Omron CX-Programmer project NewProject (CX-Programmer ?)

# PLC NewPLC1: CS1H CPU63

## Program MASTER (cyclic task 0)

### Section Section1

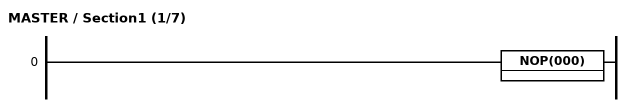
; rung 0
NOP(000)

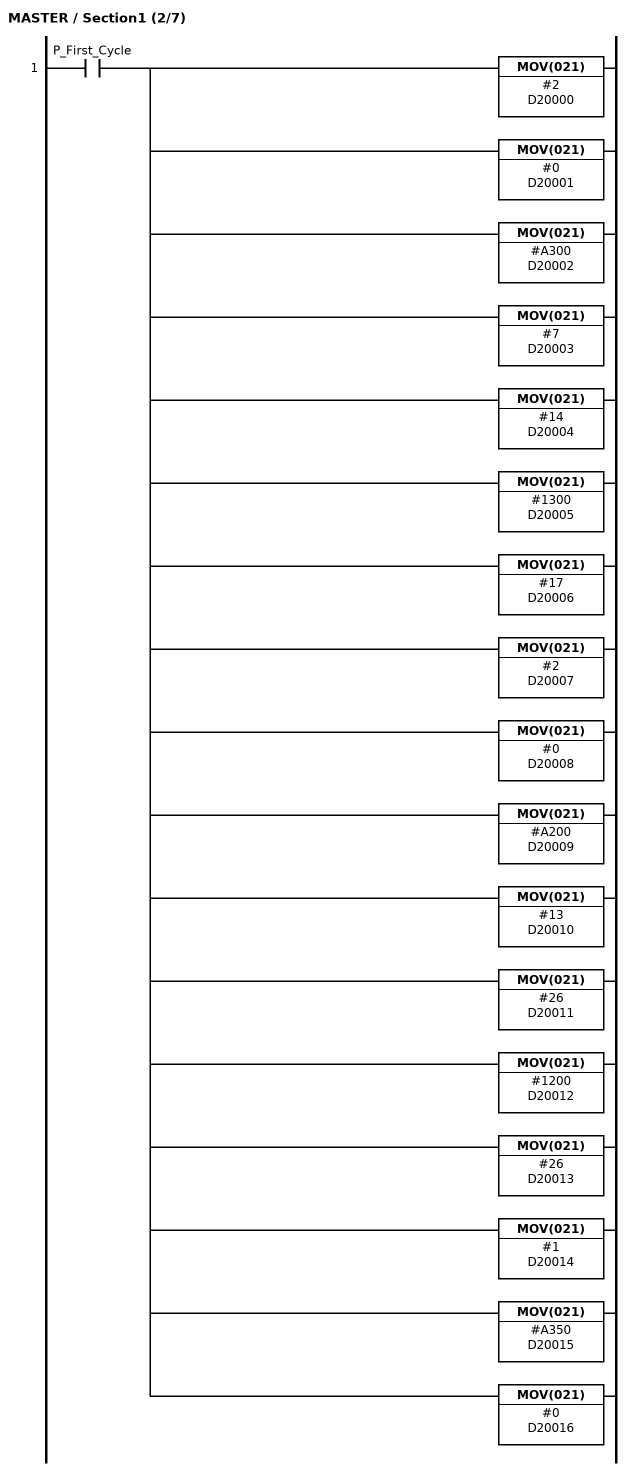
; rung 1
// R
LD P_First_Cycle  // 
MOV(021) #2 D20000
MOV(021) #0 D20001
MOV(021) #A300 D20002
MOV(021) #7 D20003
MOV(021) #14 D20004
MOV(021) #1300 D20005
MOV(021) #17 D20006
MOV(021) #2 D20007
MOV(021) #0 D20008
MOV(021) #A200 D20009
MOV(021) #13 D20010
MOV(021) #26 D20011
MOV(021) #1200 D20012
MOV(021) #26 D20013
MOV(021) #1 D20014
MOV(021) #A350 D20015
MOV(021) #0 D20016

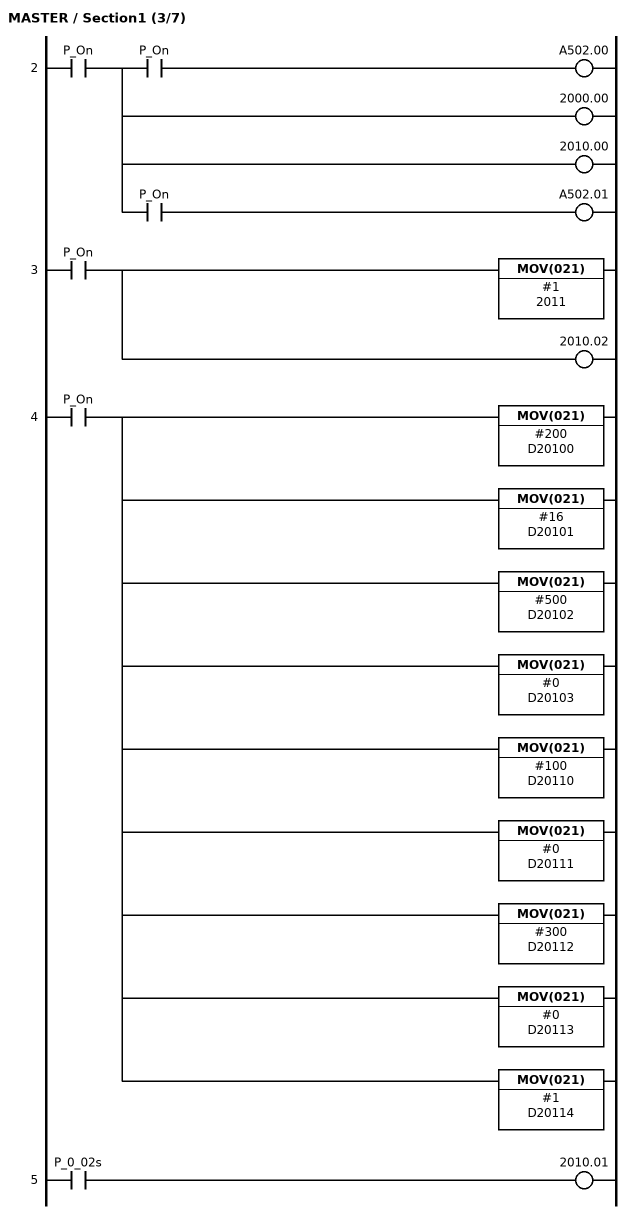
; rung 2
LD P_On
OUT TR0
AND P_On
OUT A502.00
LD TR0
OUT 2000.00
OUT 2010.00
AND P_On
OUT A502.01
; rung 3
LD P_On
MOV(021) #1 2011
OUT 2010.02
; rung 4
LD P_On
MOV(021) #200 D20100
MOV(021) #16 D20101
MOV(021) #500 D20102
MOV(021) #0 D20103
MOV(021) #100 D20110
MOV(021) #0 D20111
MOV(021) #300 D20112
MOV(021) #0 D20113
MOV(021) #1 D20114
; rung 5
LD P_0_02s
OUT 2010.01

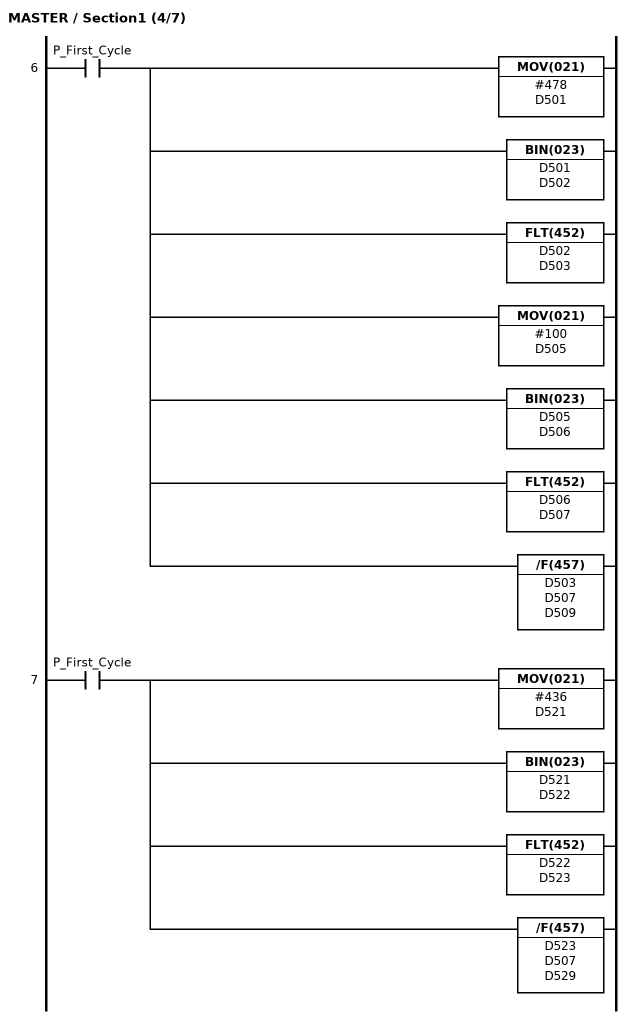
; rung 6
// R
LD P_First_Cycle
MOV(021) #478 D501
BIN(023) D501 D502
FLT(452) D502 D503
MOV(021) #100 D505
BIN(023) D505 D506
FLT(452) D506 D507
/F(457) D503 D507 D509  // 
; rung 7
// R
LD P_First_Cycle
MOV(021) #436 D521
BIN(023) D521 D522
FLT(452) D522 D523
/F(457) D523 D507 D529  // 

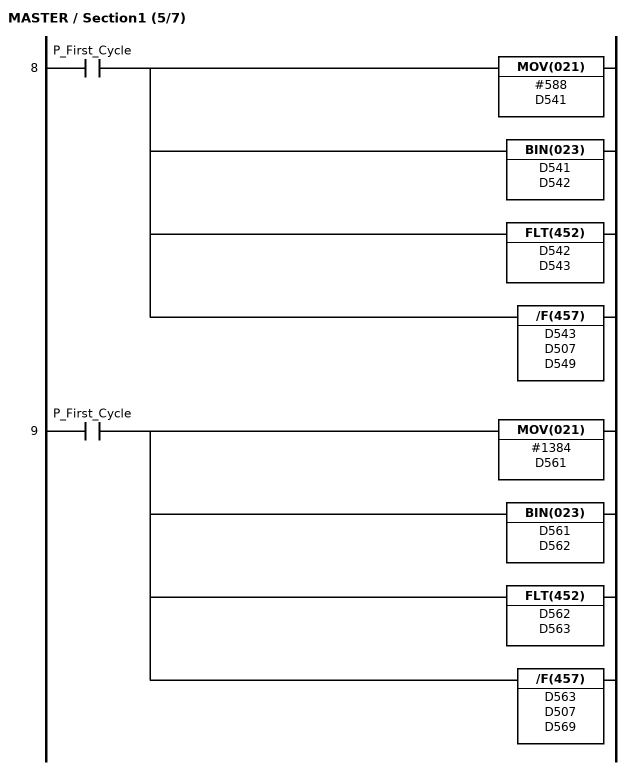
; rung 8
// R
LD P_First_Cycle
MOV(021) #588 D541
BIN(023) D541 D542
FLT(452) D542 D543
/F(457) D543 D507 D549  // 
; rung 9
// R
LD P_First_Cycle
MOV(021) #1384 D561
BIN(023) D561 D562
FLT(452) D562 D563
/F(457) D563 D507 D569  // 

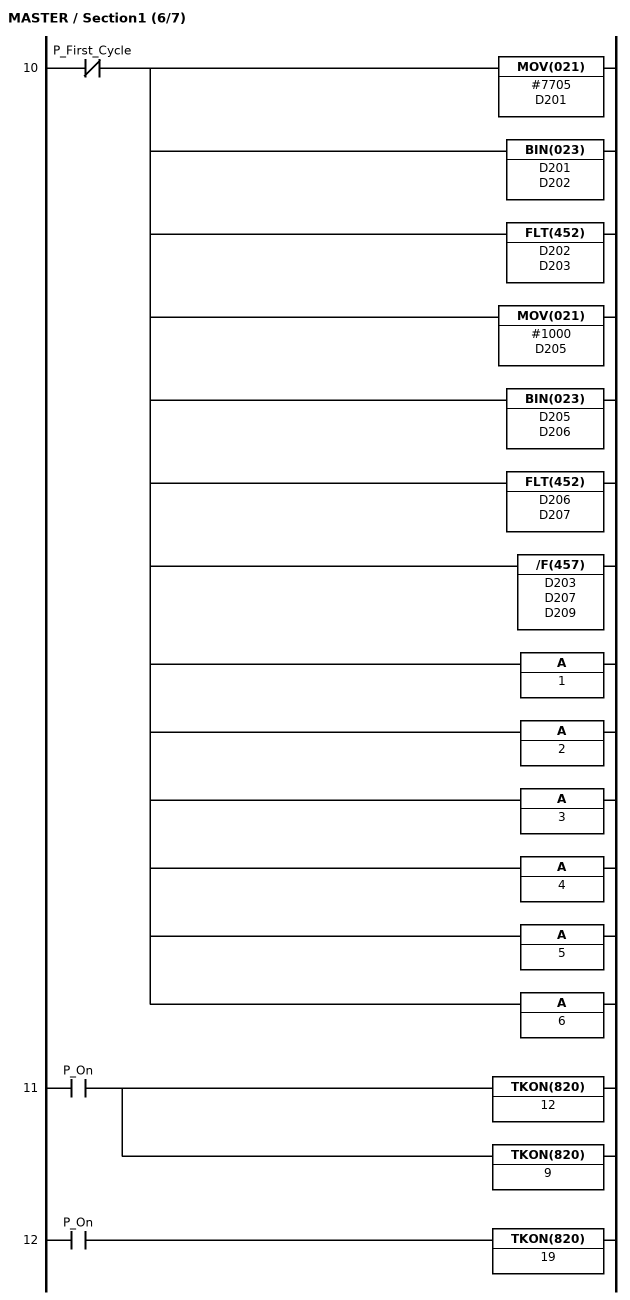
; rung 10
// R
LDNOT P_First_Cycle
MOV(021) #7705 D201
BIN(023) D201 D202
FLT(452) D202 D203
MOV(021) #1000 D205
BIN(023) D205 D206
FLT(452) D206 D207
/F(457) D203 D207 D209  // 
A  1
A  2
A  3
A  4
A  5
A  6
// 
// 
// 
// 
// 
// 
; rung 11
// R
LD P_On
TKON(820) 12
TKON(820) 9  // 
; rung 12
// R
LD P_On
TKON(820) 19  // 

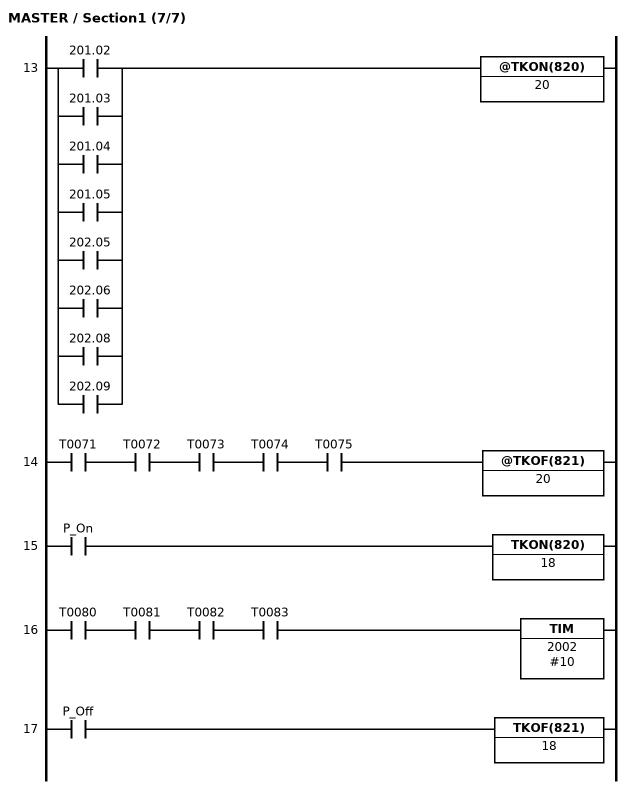
; rung 13
// R
LD 201.02
OR 201.03
OR 201.04
OR 201.05
OR 202.05
OR 202.06
OR 202.08
OR 202.09
@TKON(820) 20  // 
; rung 14
LD T0071
AND T0072
AND T0073
AND T0074
AND T0075
@TKOF(821) 20
; rung 15
// R
LD P_On
TKON(820) 18  // 
; rung 16
LD T0080
AND T0081
AND T0082
AND T0083
TIM 2002 #10
; rung 17
LD P_Off
TKOF(821) 18

### Section Section2

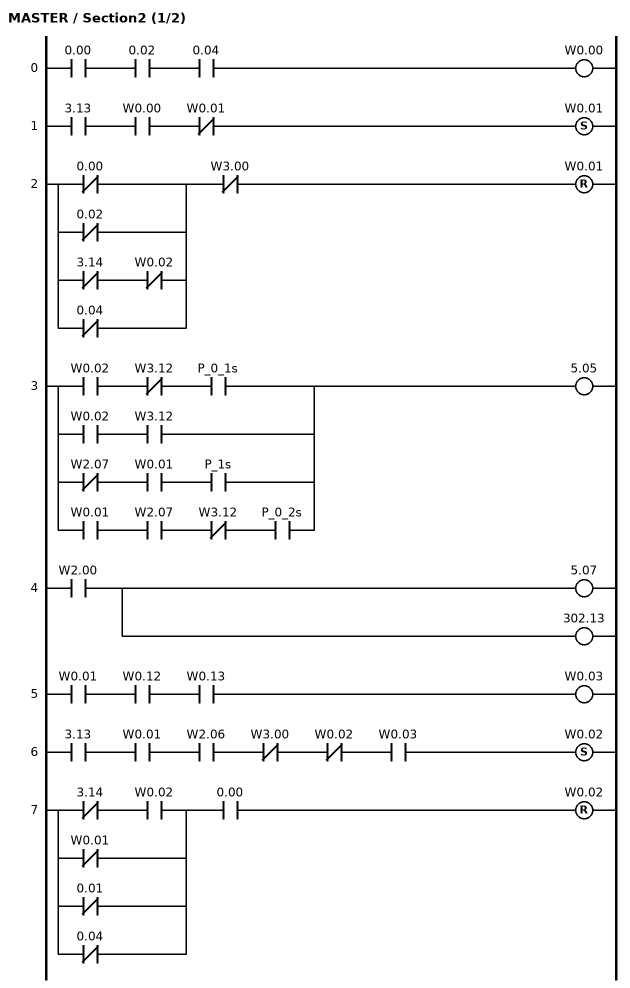
; rung 0
// R
LD 0.00
AND 0.02
AND 0.04
OUT W0.00  // 
; rung 1
LD 3.13
AND W0.00
ANDNOT W0.01
SET W0.01  // 
; rung 2
LDNOT 0.00
ORNOT 0.02
LDNOT 3.14
ANDNOT W0.02
ORLD
ORNOT 0.04
ANDNOT W3.00
RSET W0.01
; rung 3
LD W0.02
ANDNOT W3.12
AND P_0_1s
LD W0.02
AND W3.12
ORLD
LDNOT W2.07
AND W0.01
AND P_1s
ORLD
LD W0.01
AND W2.07
ANDNOT W3.12
AND P_0_2s
ORLD
OUT 5.05
; rung 4
LD W2.00
OUT 5.07
OUT 302.13
; rung 5
LD W0.01
AND W0.12
AND W0.13
OUT W0.03  // 
; rung 6
// R
LD 3.13
AND W0.01
AND W2.06
ANDNOT W3.00
ANDNOT W0.02
AND W0.03
SET W0.02
; rung 7
LDNOT 3.14
AND W0.02
ORNOT W0.01
ORNOT 0.01
ORNOT 0.04
AND 0.00
RSET W0.02

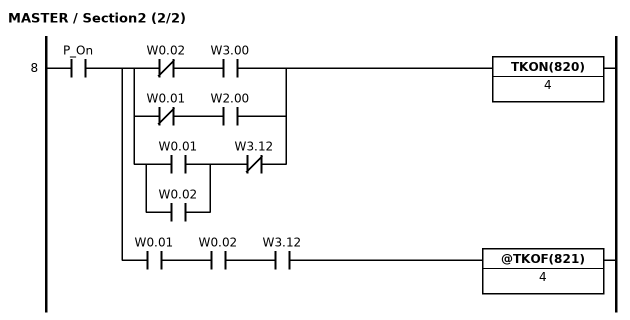
; rung 8
LD P_On
OUT TR0
LDNOT W0.02
AND W3.00
LDNOT W0.01
AND W2.00
ORLD
LD W0.01
OR W0.02
ANDNOT W3.12
ORLD
ANDLD
TKON(820) 4
LD TR0
AND W0.01
AND W0.02
AND W3.12
@TKOF(821) 4  // 

### Section Section3

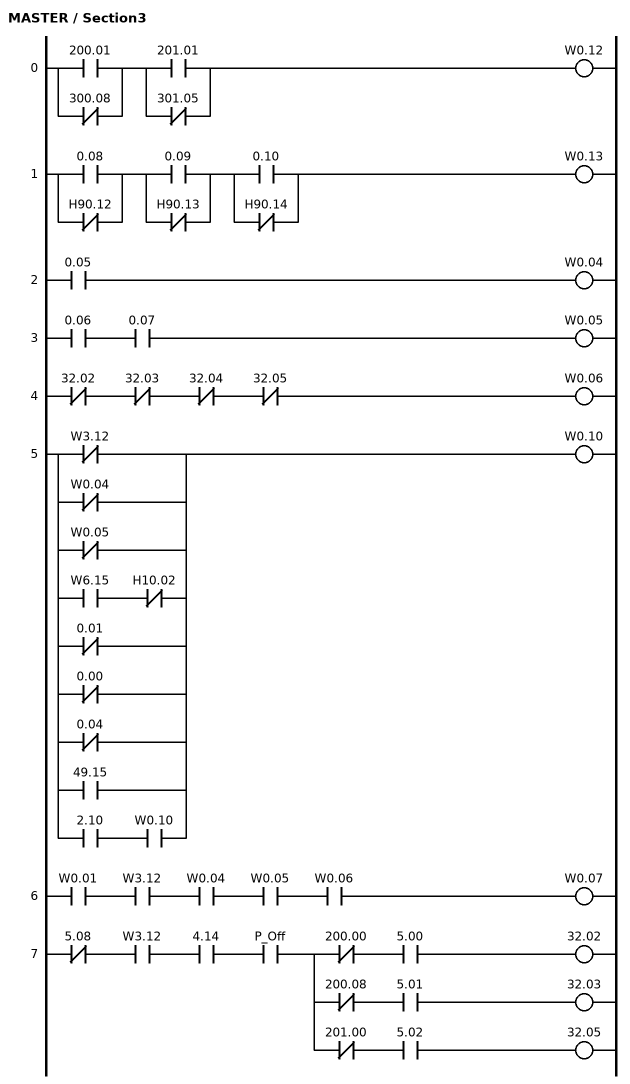
; rung 0
// R
LD 200.01
ORNOT 300.08
LD 201.01
ORNOT 301.05
ANDLD
OUT W0.12
; rung 1
LD 0.08
ORNOT H90.12
LD 0.09
ORNOT H90.13
ANDLD
LD 0.10
ORNOT H90.14
ANDLD
OUT W0.13
; rung 2
LD 0.05
OUT W0.04
; rung 3
LD 0.06
AND 0.07
OUT W0.05
; rung 4
LDNOT 32.02
ANDNOT 32.03
ANDNOT 32.04
ANDNOT 32.05
OUT W0.06
; rung 5
LDNOT W3.12
ORNOT W0.04
ORNOT W0.05
LD W6.15
ANDNOT H10.02
ORLD
ORNOT 0.01
ORNOT 0.00
ORNOT 0.04
OR 49.15
LD 2.10
AND W0.10
ORLD
OUT W0.10
; rung 6
LD W0.01
AND W3.12
AND W0.04
AND W0.05
AND W0.06
OUT W0.07
; rung 7
// R
LDNOT 5.08
AND W3.12
AND 4.14
AND P_Off
OUT TR0
ANDNOT 200.00
AND 5.00
OUT 32.02
LD TR0
ANDNOT 200.08
AND 5.01
OUT 32.03
LD TR0
ANDNOT 201.00
AND 5.02
OUT 32.05

### Section Section4

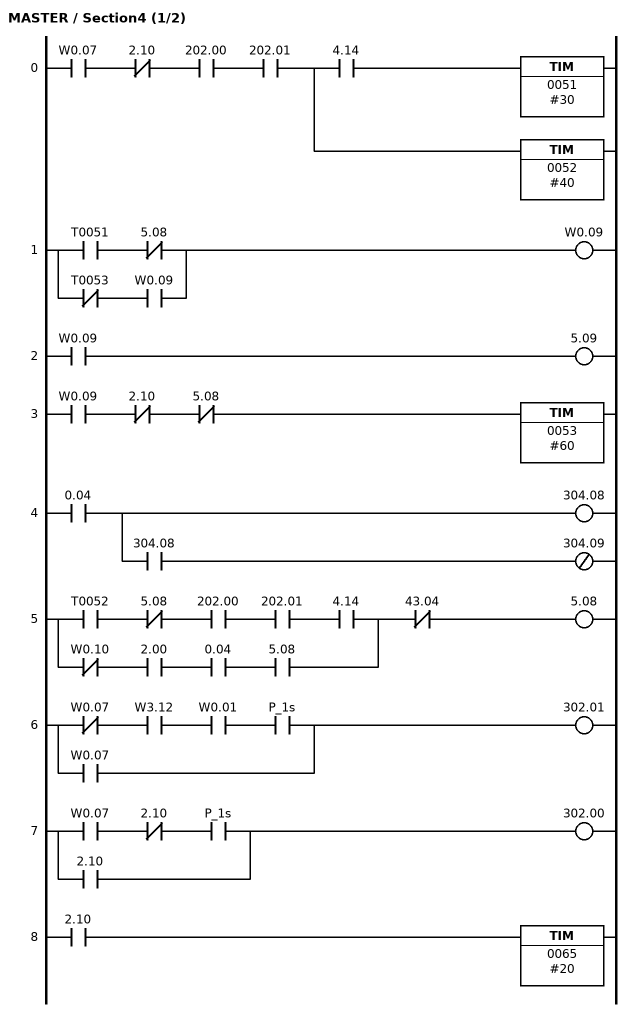
; rung 0
// R
LD W0.07
ANDNOT 2.10
AND 202.00
AND 202.01
OUT TR0
AND 4.14
TIM 0051 #30
LD TR0
TIM 0052 #40
; rung 1
LD T0051
ANDNOT 5.08
LDNOT T0053
AND W0.09
ORLD
OUT W0.09
; rung 2
LD W0.09
OUT 5.09
; rung 3
LD W0.09
ANDNOT 2.10
ANDNOT 5.08
TIM 0053 #60
; rung 4
LD 0.04
OUT 304.08
AND 304.08
OUTNOT 304.09
; rung 5
LD T0052
ANDNOT 5.08
AND 202.00
AND 202.01
AND 4.14
LDNOT W0.10
AND 2.00
AND 0.04
AND 5.08
ORLD
ANDNOT 43.04
OUT 5.08
; rung 6
LDNOT W0.07
AND W3.12
AND W0.01
AND P_1s
OR W0.07
OUT 302.01
; rung 7
LD W0.07
ANDNOT 2.10
AND P_1s
OR 2.10
OUT 302.00
; rung 8
LD 2.10
TIM 0065 #20

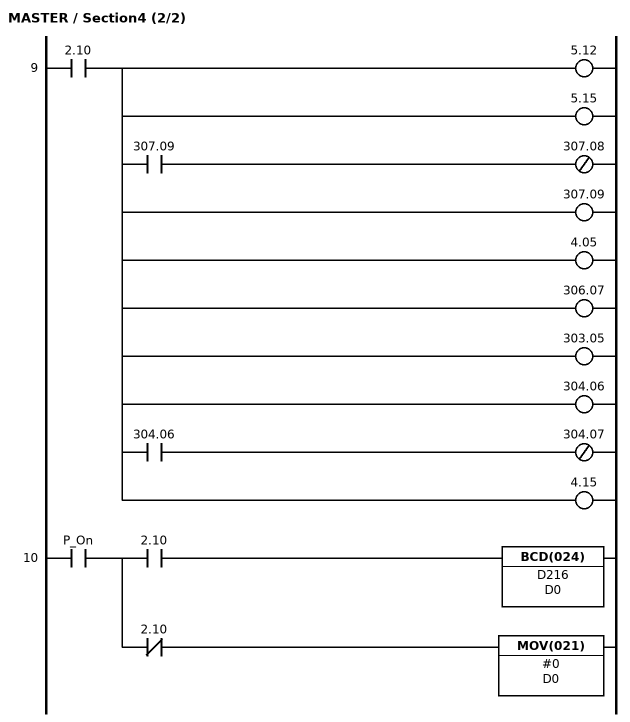
; rung 9
LD 2.10
OUT TR0
OUT 5.12
OUT 5.15
AND 307.09
OUTNOT 307.08
LD TR0
OUT 307.09
OUT 4.05
OUT 306.07
OUT 303.05
OUT 304.06
AND 304.06
OUTNOT 304.07
LD TR0
OUT 4.15
; rung 10
LD P_On
OUT TR0
AND 2.10
BCD(024) D216 D0
LD TR0
ANDNOT 2.10
MOV(021) #0 D0

### Section Section5

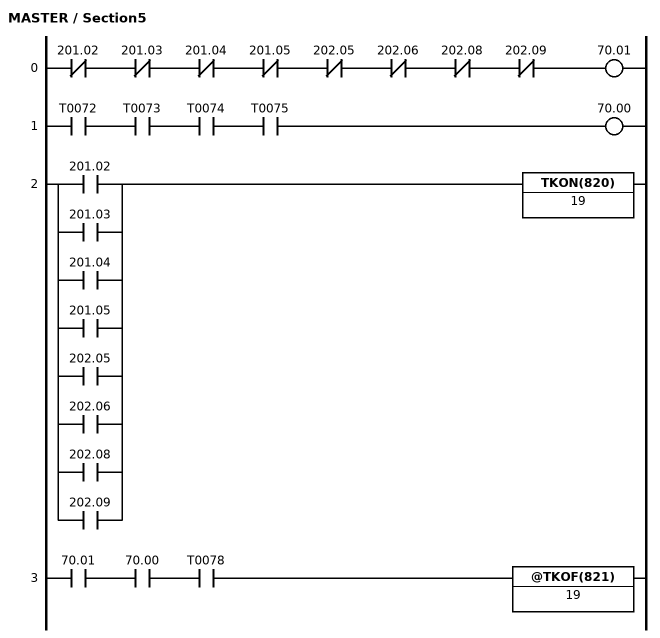
; rung 0
LDNOT 201.02
ANDNOT 201.03
ANDNOT 201.04
ANDNOT 201.05
ANDNOT 202.05
ANDNOT 202.06
ANDNOT 202.08
ANDNOT 202.09
OUT 70.01
; rung 1
LD T0072
AND T0073
AND T0074
AND T0075
OUT 70.00
; rung 2
LD 201.02
OR 201.03
OR 201.04
OR 201.05
OR 202.05
OR 202.06
OR 202.08
OR 202.09
TKON(820) 19  // 
; rung 3
LD 70.01
AND 70.00
AND T0078
@TKOF(821) 19

### Section Section6

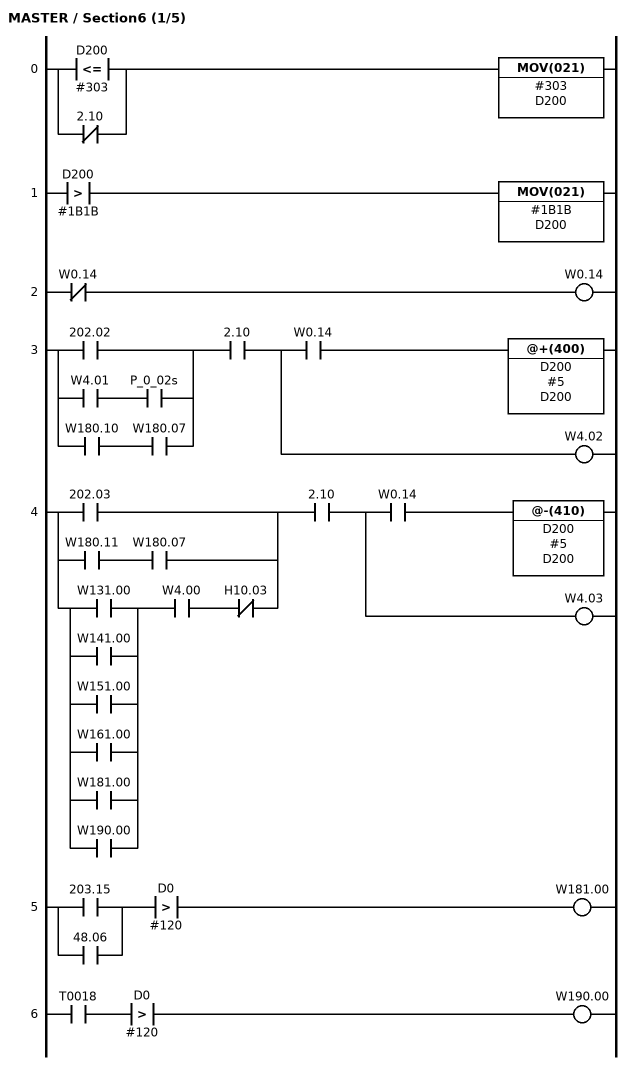
; rung 0
// R
LD<=(315) D200 #303
ORNOT 2.10
MOV(021) #303 D200  // 
; rung 1
LD>(320) D200 #1B1B
MOV(021) #1B1B D200  // 
; rung 2
LDNOT W0.14
OUT W0.14
; rung 3
// R
LD 202.02
LD W4.01
AND P_0_02s
ORLD
LD W180.10
AND W180.07
ORLD
AND 2.10
OUT TR0
AND W0.14
@+(400) D200 #5 D200
LD TR0
OUT W4.02  // 
; rung 4
// R
LD 202.03
LD W180.11
AND W180.07
ORLD
LD W131.00
OR W141.00
OR W151.00
OR W161.00
OR W181.00
OR W190.00
AND W4.00
ANDNOT H10.03
ORLD
AND 2.10
OUT TR0
AND W0.14
@-(410) D200 #5 D200
LD TR0
OUT W4.03  // 
; rung 5
// R
LD 203.15
OR 48.06
AND>(320) D0 #120
OUT W181.00
; rung 6
// R
LD T0018
AND>(320) D0 #120
OUT W190.00

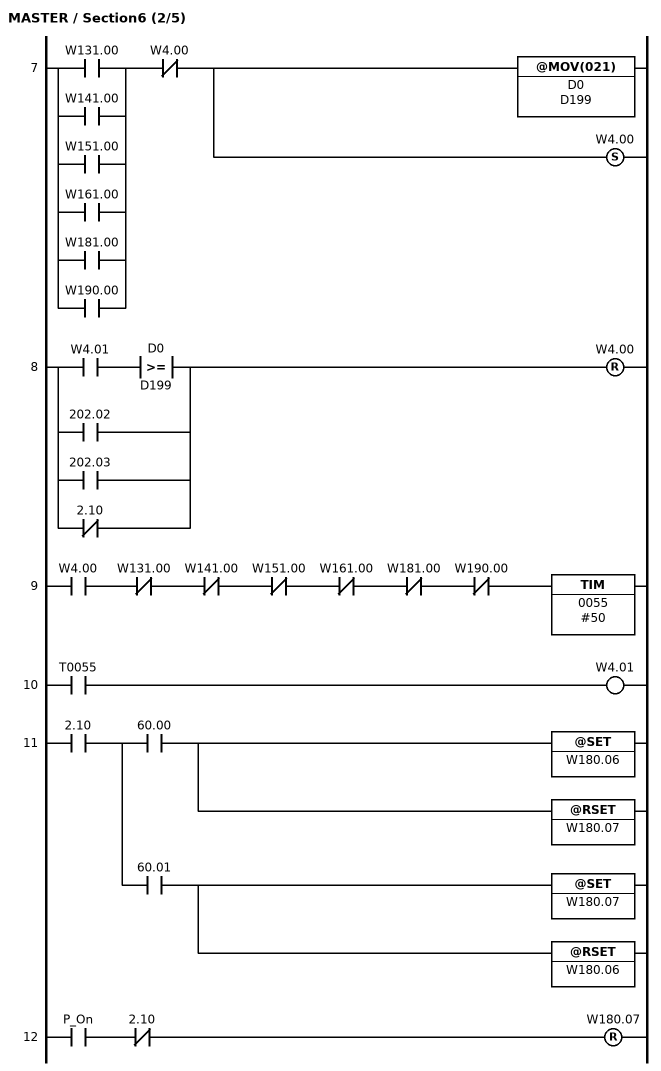
; rung 7
// R
LD W131.00
OR W141.00
OR W151.00
OR W161.00
OR W181.00
OR W190.00
ANDNOT W4.00
@MOV(021) D0 D199
SET W4.00
; rung 8
LD W4.01
AND>=(325) D0 D199
OR 202.02
OR 202.03
ORNOT 2.10
RSET W4.00
; rung 9
LD W4.00
ANDNOT W131.00
ANDNOT W141.00
ANDNOT W151.00
ANDNOT W161.00
ANDNOT W181.00
ANDNOT W190.00
TIM 0055 #50
; rung 10
LD T0055
OUT W4.01
; rung 11
LD 2.10
OUT TR0
AND 60.00
@SET W180.06
@RSET W180.07
LD TR0
AND 60.01
@SET W180.07
@RSET W180.06
; rung 12
LD P_On
ANDNOT 2.10
RSET W180.07

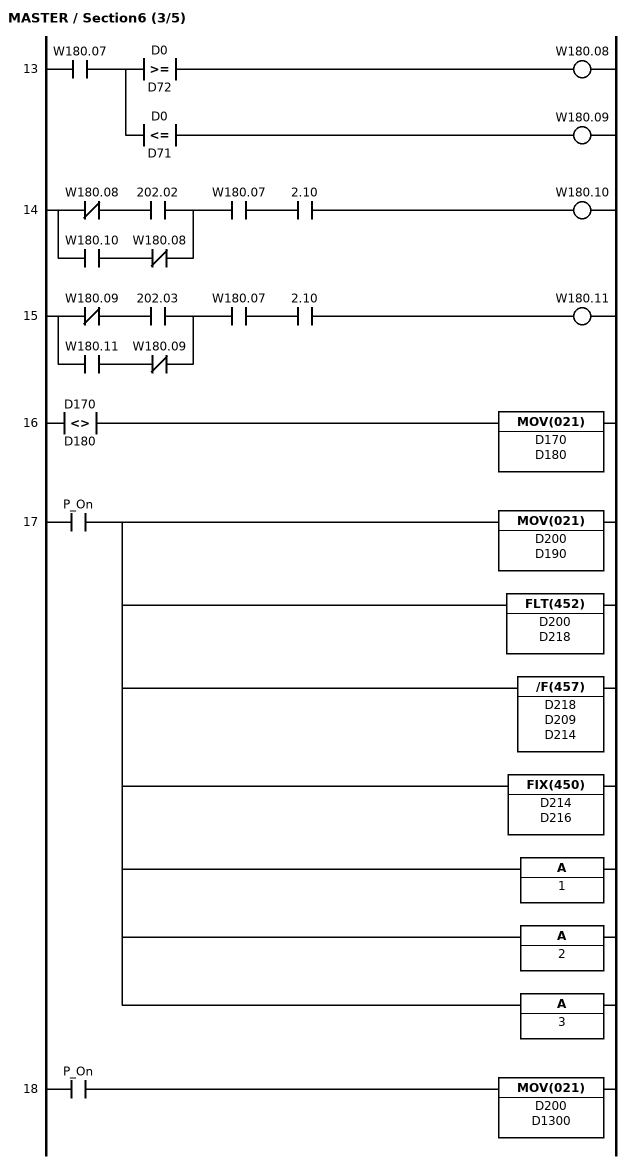
; rung 13
LD W180.07
OUT TR0
AND>=(325) D0 D72
OUT W180.08
LD TR0
AND<=(315) D0 D71
OUT W180.09
; rung 14
LDNOT W180.08
AND 202.02
LD W180.10
ANDNOT W180.08
ORLD
AND W180.07
AND 2.10
OUT W180.10
; rung 15
LDNOT W180.09
AND 202.03
LD W180.11
ANDNOT W180.09
ORLD
AND W180.07
AND 2.10
OUT W180.11
; rung 16
LD<>(305) D170 D180
MOV(021) D170 D180
; rung 17
// R
LD P_On
MOV(021) D200 D190
FLT(452) D200 D218
/F(457) D218 D209 D214
FIX(450) D214 D216  // 
A  1
A  2
A  3
// 
// 
// 
; rung 18
// R
LD P_On
MOV(021) D200 D1300

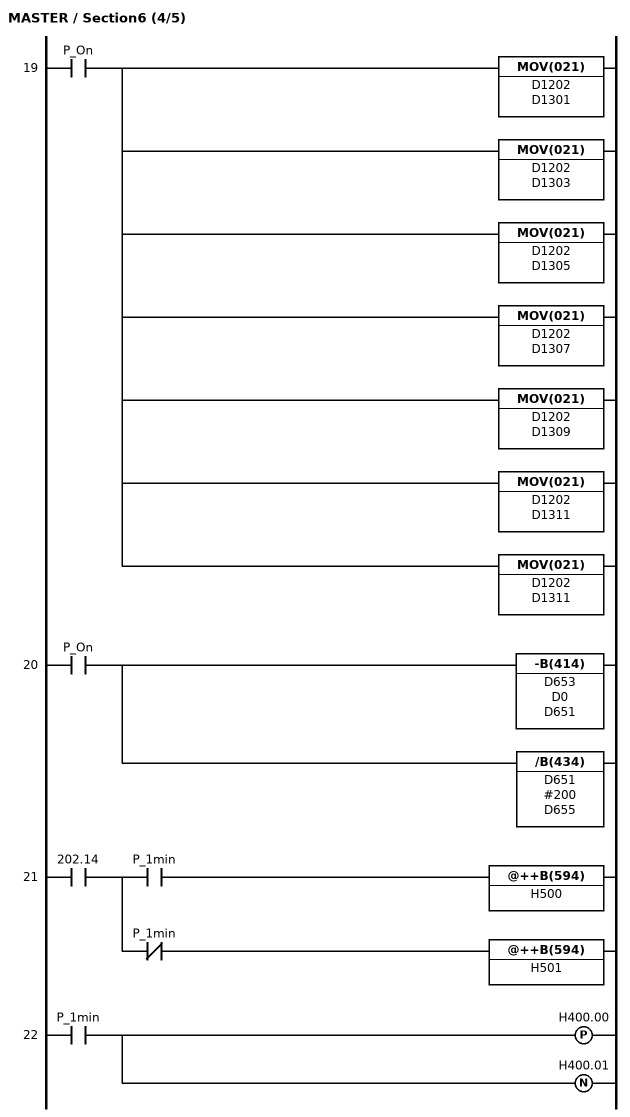
; rung 19
// R
LD P_On
MOV(021) D1202 D1301
MOV(021) D1202 D1303
MOV(021) D1202 D1305
MOV(021) D1202 D1307
MOV(021) D1202 D1309
MOV(021) D1202 D1311
MOV(021) D1202 D1311
; rung 20
LD P_On
-B(414) D653 D0 D651
/B(434) D651 #200 D655
; rung 21
// R
LD 202.14
OUT TR0
AND P_1min
@++B(594) H500
LD TR0
ANDNOT P_1min
@++B(594) H501
; rung 22
LD P_1min
DIFU(013) H400.00
DIFD(014) H400.01

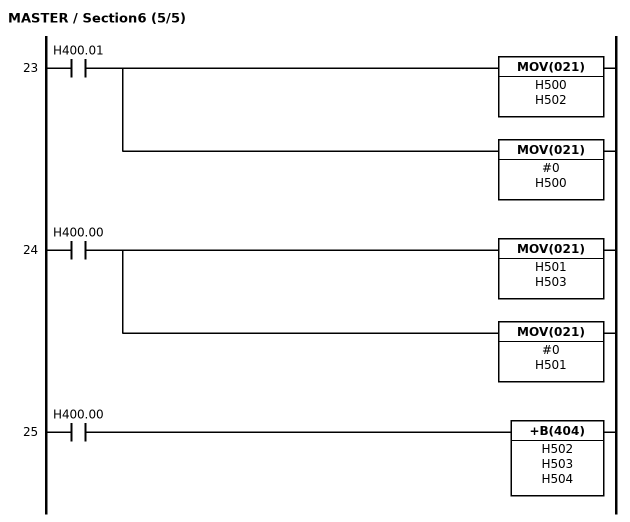
; rung 23
LD H400.01
MOV(021) H500 H502
MOV(021) #0 H500
; rung 24
LD H400.00
MOV(021) H501 H503
MOV(021) #0 H501
; rung 25
LD H400.00
+B(404) H502 H503 H504

### Section Section7

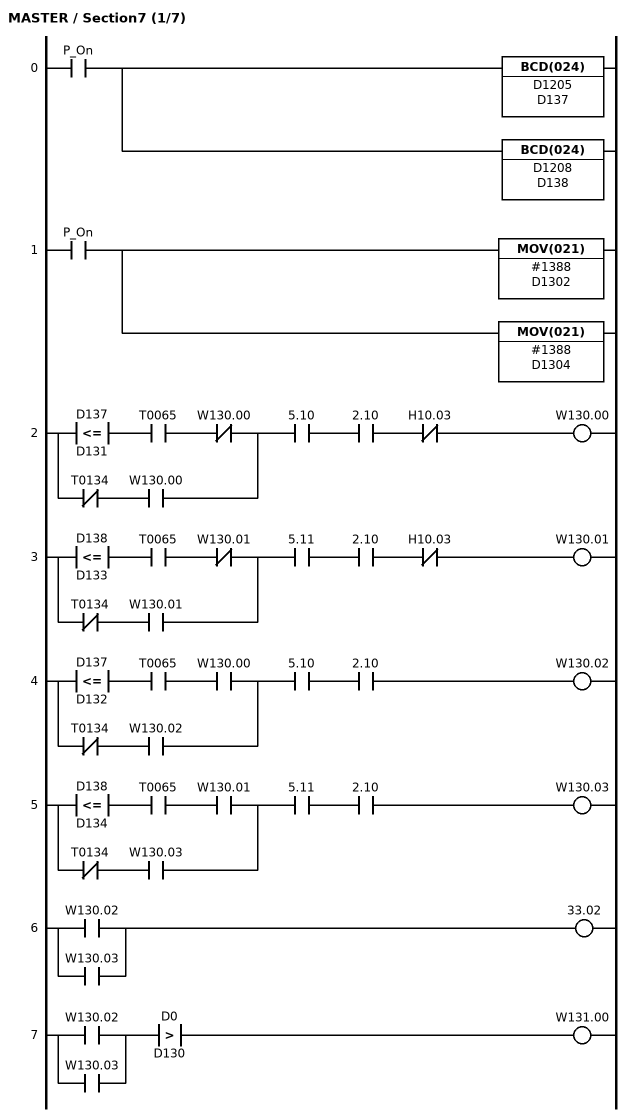
; rung 0
// R
LD P_On
BCD(024) D1205 D137
BCD(024) D1208 D138
; rung 1
// R
LD P_On
MOV(021) #1388 D1302
MOV(021) #1388 D1304
; rung 2
// R
LD<=(315) D137 D131
AND T0065
ANDNOT W130.00
LDNOT T0134
AND W130.00
ORLD
AND 5.10
AND 2.10
ANDNOT H10.03
OUT W130.00
; rung 3
LD<=(315) D138 D133
AND T0065
ANDNOT W130.01
LDNOT T0134
AND W130.01
ORLD
AND 5.11
AND 2.10
ANDNOT H10.03
OUT W130.01
; rung 4
LD<=(315) D137 D132
AND T0065
AND W130.00
LDNOT T0134
AND W130.02
ORLD
AND 5.10
AND 2.10
OUT W130.02
; rung 5
LD<=(315) D138 D134
AND T0065
AND W130.01
LDNOT T0134
AND W130.03
ORLD
AND 5.11
AND 2.10
OUT W130.03
; rung 6
LD W130.02
OR W130.03
OUT 33.02
; rung 7
// R
LD W130.02
OR W130.03
AND>(320) D0 D130
OUT W131.00

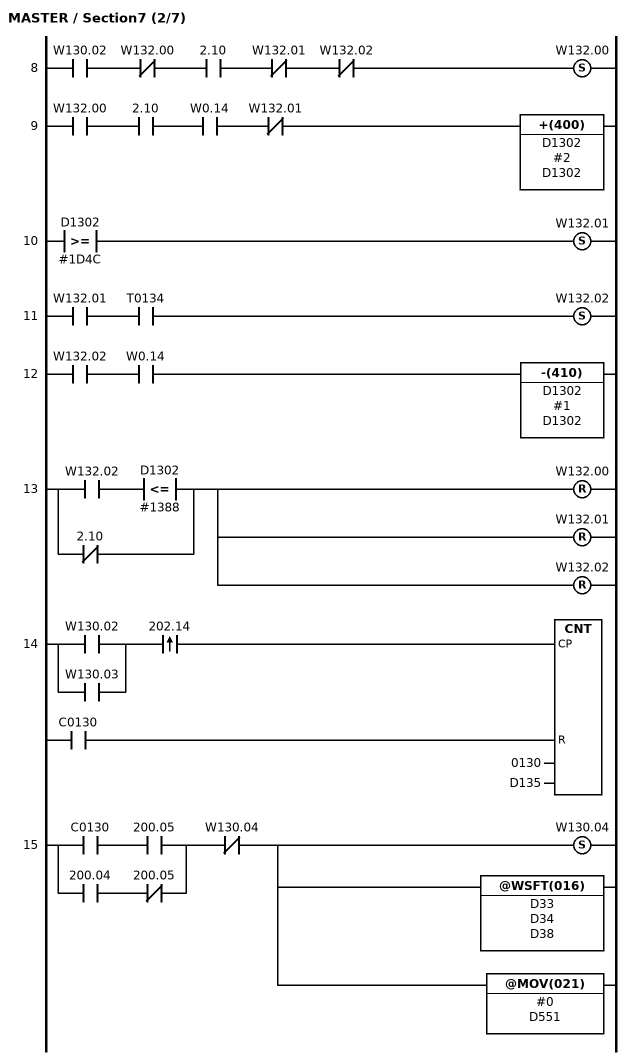
; rung 8
LD W130.02
ANDNOT W132.00
AND 2.10
ANDNOT W132.01
ANDNOT W132.02
SET W132.00
; rung 9
LD W132.00
AND 2.10
AND W0.14
ANDNOT W132.01
+(400) D1302 #2 D1302
; rung 10
LD>=(325) D1302 #1D4C
SET W132.01
; rung 11
LD W132.01
AND T0134
SET W132.02
; rung 12
LD W132.02
AND W0.14
-(410) D1302 #1 D1302
; rung 13
LD W132.02
AND<=(315) D1302 #1388
ORNOT 2.10
RSET W132.00
RSET W132.01
RSET W132.02
; rung 14
LD W130.02
OR W130.03
@AND 202.14
LD C0130
CNT 0130 D135
; rung 15
LD C0130
AND 200.05
LD 200.04
ANDNOT 200.05
ORLD
ANDNOT W130.04
SET W130.04
@WSFT(016) D33 D34 D38
@MOV(021) #0 D551

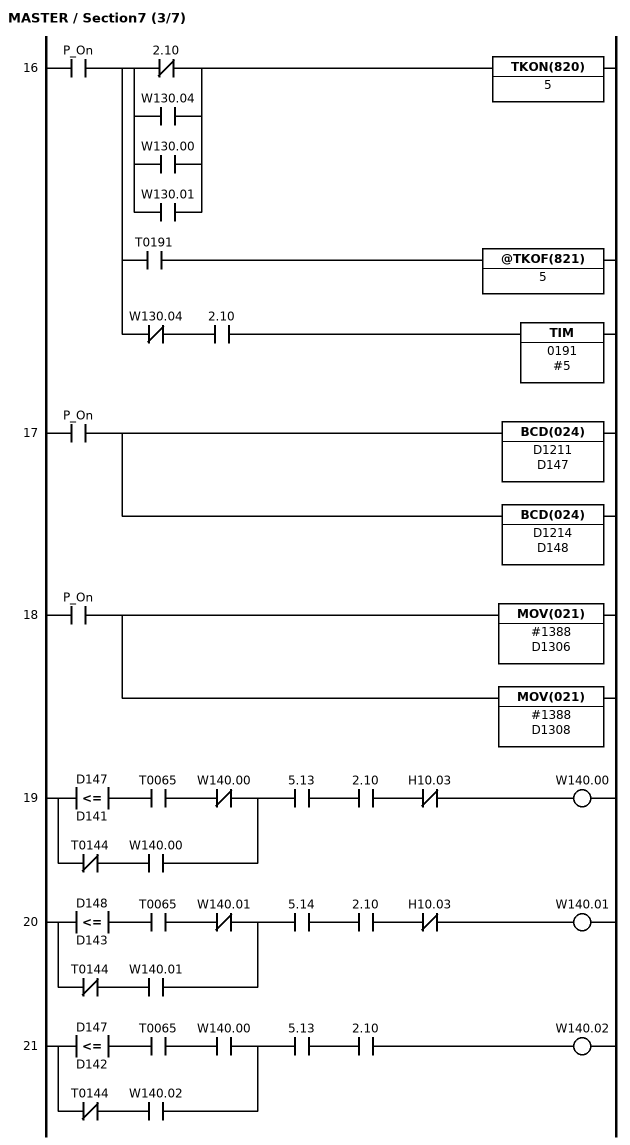
; rung 16
LD P_On
OUT TR0
LDNOT 2.10
OR W130.04
OR W130.00
OR W130.01
ANDLD
TKON(820) 5
LD TR0
AND T0191
@TKOF(821) 5
LD TR0
ANDNOT W130.04
AND 2.10
TIM 0191 #5  // 
; rung 17
// R
LD P_On
BCD(024) D1211 D147
BCD(024) D1214 D148
; rung 18
// R
LD P_On
MOV(021) #1388 D1306
MOV(021) #1388 D1308
; rung 19
// R
LD<=(315) D147 D141
AND T0065
ANDNOT W140.00
LDNOT T0144
AND W140.00
ORLD
AND 5.13
AND 2.10
ANDNOT H10.03
OUT W140.00
; rung 20
LD<=(315) D148 D143
AND T0065
ANDNOT W140.01
LDNOT T0144
AND W140.01
ORLD
AND 5.14
AND 2.10
ANDNOT H10.03
OUT W140.01
; rung 21
LD<=(315) D147 D142
AND T0065
AND W140.00
LDNOT T0144
AND W140.02
ORLD
AND 5.13
AND 2.10
OUT W140.02

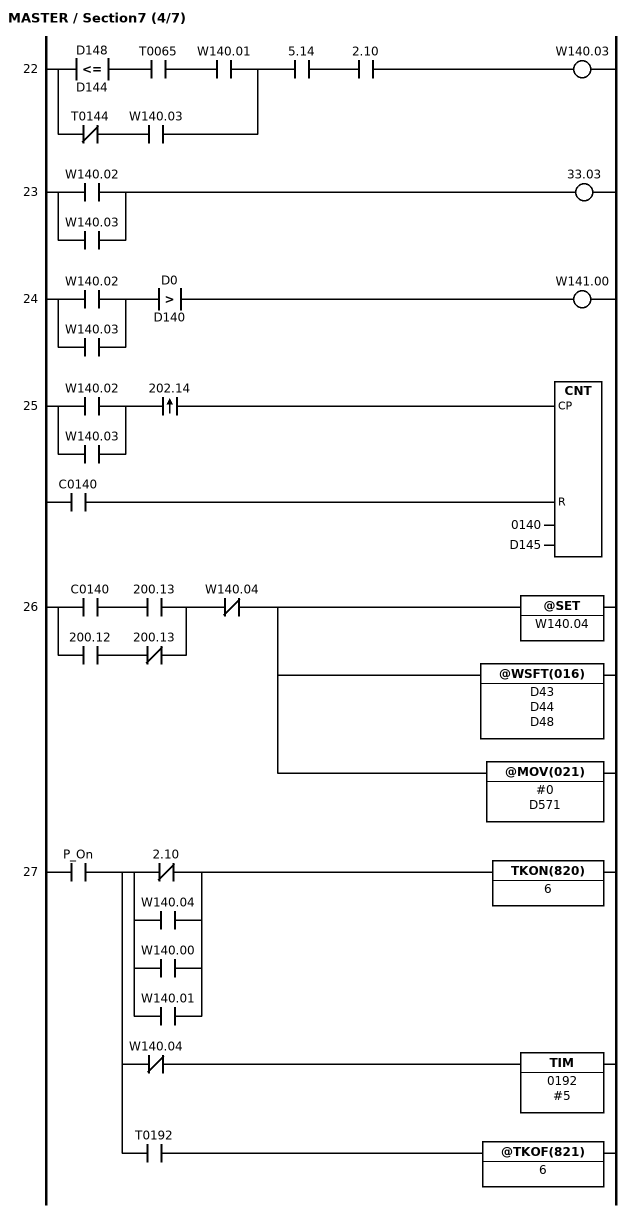
; rung 22
LD<=(315) D148 D144
AND T0065
AND W140.01
LDNOT T0144
AND W140.03
ORLD
AND 5.14
AND 2.10
OUT W140.03
; rung 23
LD W140.02
OR W140.03
OUT 33.03
; rung 24
// R
LD W140.02
OR W140.03
AND>(320) D0 D140
OUT W141.00
; rung 25
LD W140.02
OR W140.03
@AND 202.14
LD C0140
CNT 0140 D145
; rung 26
LD C0140
AND 200.13
LD 200.12
ANDNOT 200.13
ORLD
ANDNOT W140.04
@SET W140.04
@WSFT(016) D43 D44 D48
@MOV(021) #0 D571
; rung 27
LD P_On
OUT TR0
LDNOT 2.10
OR W140.04
OR W140.00
OR W140.01
ANDLD
TKON(820) 6
LD TR0
ANDNOT W140.04
TIM 0192 #5
LD TR0
AND T0192
@TKOF(821) 6  // 

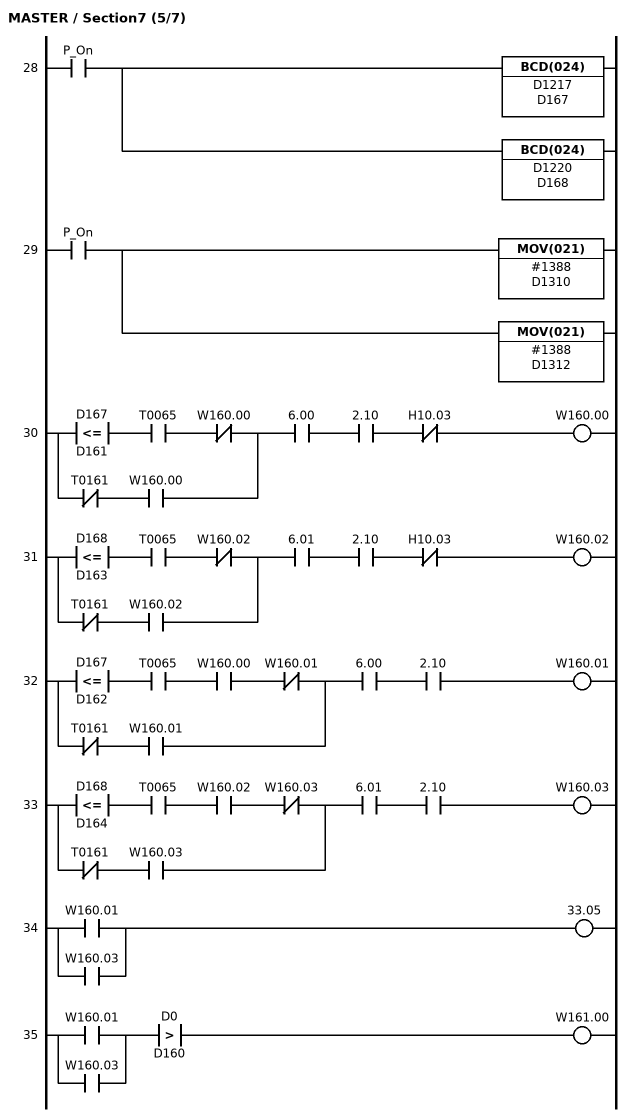
; rung 28
// R
LD P_On
BCD(024) D1217 D167
BCD(024) D1220 D168
; rung 29
// R
LD P_On
MOV(021) #1388 D1310
MOV(021) #1388 D1312
; rung 30
// R
LD<=(315) D167 D161
AND T0065
ANDNOT W160.00
LDNOT T0161
AND W160.00
ORLD
AND 6.00
AND 2.10
ANDNOT H10.03
OUT W160.00
; rung 31
// R
LD<=(315) D168 D163
AND T0065
ANDNOT W160.02
LDNOT T0161
AND W160.02
ORLD
AND 6.01
AND 2.10
ANDNOT H10.03
OUT W160.02
; rung 32
LD<=(315) D167 D162
AND T0065
AND W160.00
ANDNOT W160.01
LDNOT T0161
AND W160.01
ORLD
AND 6.00
AND 2.10
OUT W160.01
; rung 33
LD<=(315) D168 D164
AND T0065
AND W160.02
ANDNOT W160.03
LDNOT T0161
AND W160.03
ORLD
AND 6.01
AND 2.10
OUT W160.03
; rung 34
LD W160.01
OR W160.03
OUT 33.05
; rung 35
// R
LD W160.01
OR W160.03
AND>(320) D0 D160
OUT W161.00

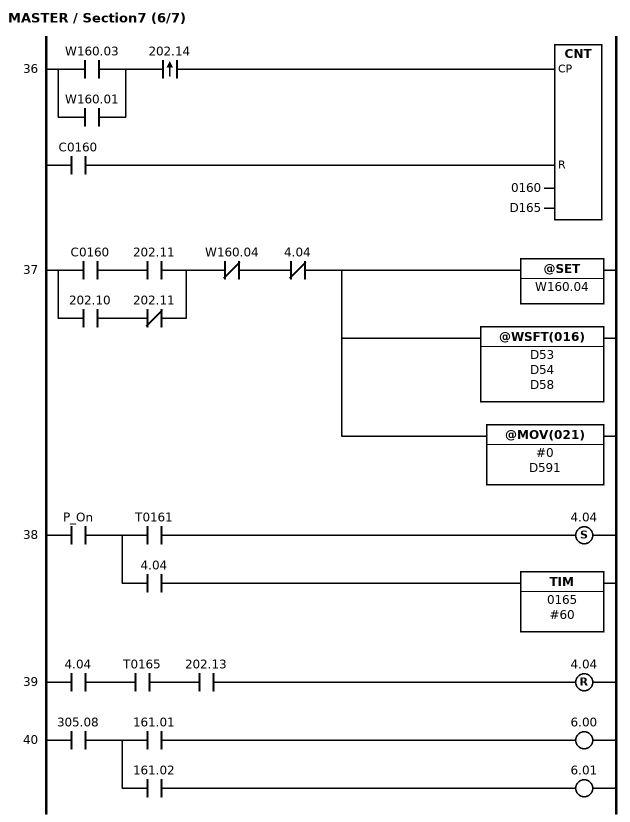
; rung 36
LD W160.03
OR W160.01
@AND 202.14
LD C0160
CNT 0160 D165
; rung 37
LD C0160
AND 202.11
LD 202.10
ANDNOT 202.11
ORLD
ANDNOT W160.04
ANDNOT 4.04
@SET W160.04
@WSFT(016) D53 D54 D58
@MOV(021) #0 D591
; rung 38
LD P_On
OUT TR0
AND T0161
SET 4.04
LD TR0
AND 4.04
TIM 0165 #60
; rung 39
LD 4.04
AND T0165
AND 202.13
RSET 4.04
; rung 40
LD 305.08
OUT TR0
AND 161.01
OUT 6.00
LD TR0
AND 161.02
OUT 6.01

